Yaskawa INFORM job: TEST_R2_NEW.JBI

/JOB
//NAME TEST_R2_NEW
///FOLDERNAME INNE
//POS
///NPOS 3,3,3,0,0,0
///TOOL 0
///POSTYPE PULSE
///PULSE
C00000=128904,5514,-49112,72908,68146,-61056
C00001=208342,-104666,-113843,10386,19704,-41798
C00002=120725,26713,56510,51500,52607,77760
BC00000=263110,-108033,800405
BC00001=336112,59246,800405
BC00002=368716,46082,571804
EC00000=0,0
EC00001=0,0
EC00002=0,0
//INST
///DATE 2023/11/01 18:40
///ATTR SC,RW
///GROUP1 RB1,BS1
///GROUP2 ST1
NOP
'test_r2_new
MOVJ C00000 BC00000 VJ=100.00  +MOVJ EC00000 VJ=100.00
MOVJ C00001 BC00001 VJ=100.00  +MOVJ EC00001 VJ=100.00
MOVJ C00002 BC00002 VJ=100.00  +MOVJ EC00002 VJ=100.00
END
